// TwinCAT 3 PLC project PLC
// ProgramVersion: 3.1.4024.0
// libraries:
//   CmpBitmapPool, * (System)
//   Tc2_Standard, * (Beckhoff Automation GmbH)
//   Tc2_System, * (Beckhoff Automation GmbH)
//   Tc3_Module, * (Beckhoff Automation GmbH)
//   VisuDialogs, * (System)
//   VisuSymbols,3.5.10.0,System
// project tree:
//   DUTs/ CarPos.TcDUT
//   / GlobalTextList.TcGTLO, PlcTask.TcTTO
//   GVLs/ GVL.TcGVL
//   POUs/ CarHandle.TcPOU, MAIN.TcPOU
//   VISUs/ ImagePool.TcIPO (not stored), Visualization Manager.TcVMO (not stored), Visualization.TcVIS
// real-time tasks:
//   TASK PlcTask: cycle T#10ms, priority 20, ADS port 350

CONFIGURATION PLC
    RESOURCE PLC ON TwinCAT3
        TASK PlcTask(INTERVAL := T#10ms, PRIORITY := 20);
        PROGRAM MAIN WITH PlcTask : MAIN;
    END_RESOURCE
END_CONFIGURATION

// ---- DUTs/CarPos.TcDUT
TYPE CarPos :
STRUCT
// coordinates of car position in 3d parking
	X:	INT;
	Y:	INT;
	Z:	INT;
END_STRUCT
END_TYPE

// ---- GVLs/GVL.TcGVL
{attribute 'qualified_only'}
VAR_GLOBAL CONSTANT
	XPosMax		:	WORD:=2;
	YPosMax		:	WORD:=3;
	ZPosMax		:	WORD:=4;
END_VAR

// ---- POUs/MAIN.TcPOU
PROGRAM MAIN
VAR
	CarPlates		:	ARRAY [1..24] OF STRING(15) := ['AB12345', 'CD98765', 'EF24689', 'GH88888', 'IJ33388',
														'KL57483', 'MN35991', 'OP46819', 'RS00001', 'TU22229',
														'DE13578', 'ZX90909', 'YW10101', 'VW46372', 'ZZ00220',
														'WE00772', 'JK77001', 'PO39120', 'LW09126', 'RM01928',
														'EK11998', 'WY00664', 'HS05524', 'TT00099'];

	InsertCar		:	BOOL;					// insert car trigger
	
	FindCar			:	BOOL;					// find car trigger
	PlateToFind		:	STRING(15);				// car plate which should be found in the car park
	CarFoundPos		:	CarPos;					// position of found car
	
	RemoveCar		:	BOOL;					// remove car trigger
	CarToRemove		:	STRING(15);				// car plate which should be removed from the car park
	
	GetNoFreePlaces	:	BOOL;					// trigger for getting number of free places in car park
	
	rtAction		:	ARRAY[1..5] OF R_TRIG;
	FreePlaces		:	INT;
	
	CarHandle		:	CarHandle;
	
	Result			: 	BOOL;					// operation result
END_VAR

VAR RETAIN PERSISTENT
	CarPark			: ARRAY [1..GVL.XPosMax, 1..GVL.YPosMax, 1..GVL.ZPosMax] OF STRING(15);
	Idx				:	INT:=1;
END_VAR

CarHandle(ArrayPark:=CarPark);


rtAction[1](CLK:=InsertCar);
rtAction[2](CLK:=FindCar);
rtAction[3](CLK:=RemoveCar);
rtAction[4](CLK:=GetNoFreePlaces);

// insert car
IF rtAction[1].Q THEN
	Result := CarHandle.M_InsertCar(CarPlates[Idx]);
	FreePlaces := CarHandle.P_NumberFreePositions;
	Idx:= Idx + 1;
	IF Idx > 24 THEN 
		Idx := 1;
	END_IF
END_IF

// find car
IF rtAction[2].Q THEN
	Result := CarHandle.M_FindCar(CarPlate:=PlateToFind,FoundCarPos=>CarFoundPos);
END_IF

// delete car
IF rtAction[3].Q THEN
	Result := CarHandle.M_RemoveCar(CarPlate := CarToRemove);
	FreePlaces := CarHandle.P_NumberFreePositions;
END_IF

// get number of free places in car park
IF rtAction[4].Q THEN
	FreePlaces := CarHandle.P_NumberFreePositions;
END_IF

END_PROGRAM

// ---- POUs/CarHandle.TcPOU
FUNCTION_BLOCK CarHandle
VAR_INPUT
END_VAR
VAR_OUTPUT
END_VAR
VAR_IN_OUT
	ArrayPark		:	ARRAY[*,*,*] OF STRING(15);	// pointer to 3d array
END_VAR
VAR
	Loop			:	CarPos;						// temp. variable
	TotalPositions	: 	INT;						// total number of car positions in car park
END_VAR

(*
This FB handles three dimensional car park.
- ArrayPark - Dimension of the car park
*)


// copy ARRAY to local variables
Loop.X := DINT_TO_INT(UPPER_BOUND(ArrayPark,1));		// cordinate X
Loop.Y := DINT_TO_INT(UPPER_BOUND(ArrayPark,2));		// cordinate Y
Loop.Z := DINT_TO_INT(UPPER_BOUND(ArrayPark,3));		// cordinate Z

// total number of car positions in car park
TotalPositions := Loop.X * Loop.Y * Loop.Z;

METHOD M_FindCar : BOOL
VAR_INPUT
	CarPlate		:	STRING(15);		// plate number of the car
END_VAR
VAR
	CarPos			:	CarPos;			// location in car park
END_VAR
VAR_OUTPUT
	FoundCarPos		:	CarPos;			// location in car park
END_VAR
(*
This Method finds car in car park using its car plate.
CarPlate - car number plate which should be looked for in car park
Methods Returns TRUE if car was successfully found, otherwise FALSE
*)

// Loop over all position in the 3D car park
FOR CarPos.X:=1 TO Loop.X DO
	FOR CarPos.Y:=1 TO Loop.Y DO
		FOR CarPos.Z:=1 TO Loop.Z DO
			
			IF  FIND(ArrayPark[CarPos.X, CarPos.Y, CarPos.Z], CarPlate) > 0 THEN
				FoundCarPos := CarPos;	// copy coordinates where car was located
				M_FindCar := TRUE;
				RETURN;
			END_IF
			
		END_FOR
	END_FOR
END_FOR
M_FindCar := FALSE;
END_METHOD

METHOD M_InsertCar : BOOL
VAR_INPUT
	CarPlate		:	STRING(15);		// plate number of the car
END_VAR
VAR
	CarPos			:	CarPos;			// location in car park
END_VAR
(*
This Method inserts one car into car park.
CarPlate - car number plate which should be insert into car park
Methods Returns TRUE if car was successfully inserted, otherwise FALSE
*)

// Loop over all position in the 3D car park
FOR CarPos.X:=1 TO Loop.X DO
	FOR CarPos.Y:=1 TO Loop.Y DO
		FOR CarPos.Z:=1 TO Loop.Z DO
			
			// insert car at the first free location in the car park
			IF ArrayPark[CarPos.X, CarPos.Y, CarPos.Z]='' THEN
				ArrayPark[CarPos.X, CarPos.Y, CarPos.Z] := CarPlate;
				M_InsertCar := TRUE;
				RETURN;
			END_IF
			
		END_FOR
	END_FOR
END_FOR

M_InsertCar := FALSE;
END_METHOD

METHOD M_RemoveCar : BOOL
VAR_INPUT
	CarPlate		:	STRING(15);		// plate number of the car
END_VAR

VAR
	CarPos			:	CarPos;			// location in car park
END_VAR
(*
This Method removes one car in car park.
CarPlate - car number plate which should be removed in car park
Methods Returns TRUE if car was successfully removed, otherwise FALSE
*)

// Loop over all position in the 3D car park
FOR CarPos.X:=1 TO Loop.X DO
	FOR CarPos.Y:=1 TO Loop.Y DO
		FOR CarPos.Z:=1 TO Loop.Z DO
			
				IF FIND(ArrayPark[CarPos.X, CarPos.Y, CarPos.Z], CarPlate) > 0 THEN
					ArrayPark[CarPos.X, CarPos.Y, CarPos.Z]:=''; 	// remove car = set string empty 
					M_RemoveCar := TRUE;
					RETURN;
				END_IF
			
		END_FOR
	END_FOR
END_FOR

M_RemoveCar := TRUE;
END_METHOD

PROPERTY P_NumberFreePositions : INT

// Property returns number of free locations in car park
GET
VAR
	CarCount		: 	INT;			// number of occupied par places in car park
	CarPos			:	CarPos;			// location in car park
END_VAR
// Loop over all position in the 3D car park
FOR CarPos.X:=1 TO Loop.X DO
	FOR CarPos.Y:=1 TO Loop.Y DO
		FOR CarPos.Z:=1 TO Loop.Z DO
			
			IF ArrayPark[CarPos.X, CarPos.Y, CarPos.Z] <> '' THEN
				CarCount := CarCount+1;
			END_IF
			
		END_FOR
	END_FOR
END_FOR

P_NumberFreePositions := TotalPositions - CarCount;
END_GET
END_PROPERTY

END_FUNCTION_BLOCK

// ---- GlobalTextList.TcGTLO
TEXTLIST GlobalTextList
  316 = '%s'
  656 = '12387812'
  188 = 'Car Plate to Delete:'
  264 = 'Car PLate to Find:'
  432 = 'Car Plate to Find:'
  625 = 'Car to delete'
  296 = 'Car to Delete:'
  833 = 'Car to remove'
  597 = 'Car to Remove:'
  485 = 'Delete Car'
  174 = 'Find Car'
  267 = 'Found Car Position'
  242 = 'Insert Car'
  115 = 'Label'
  455 = 'Number of free places:\n\n%d'
  904 = 'Number of free places:\n%d'
  459 = 'Plate to delete'
  778 = 'Plate to find'
  298 = 'Plate to find: %s'
  396 = 'Remove Car'
  783 = 'Three Dimension Car Park'
  877 = 'X'
  615 = 'Y'
  950 = 'Z'
END_TEXTLIST

// ---- VISUs/Visualization.TcVIS
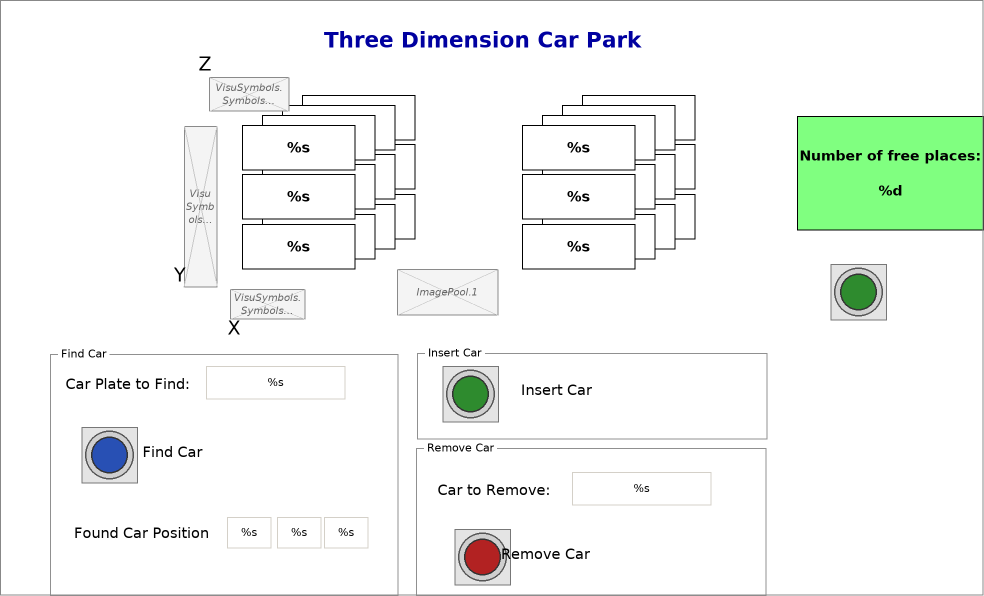
VISUALIZATION Visualization  // 984x596
    Rectangle (302,95 113x45), "%s", text variable: MAIN.CarPark[1,3,4], colour toggle: MAIN.CarPark[1,3,4] <> ''
    Rectangle (302,194 113x45), "%s", text variable: MAIN.CarPark[1,1,4], colour toggle: MAIN.CarPark[1,1,4] <> ''
    Rectangle (302,144 113x45), "%s", text variable: MAIN.CarPark[1,2,4], colour toggle: MAIN.CarPark[1,2,4] <> ''
    Rectangle (282,204 113x45), "%s", text variable: MAIN.CarPark[1,1,3], colour toggle: MAIN.CarPark[1,1,3] <> ''
    Rectangle (282,154 113x45), "%s", text variable: MAIN.CarPark[1,2,3], colour toggle: MAIN.CarPark[1,2,3] <> ''
    Rectangle (282,105 113x45), "%s", text variable: MAIN.CarPark[1,3,3], colour toggle: MAIN.CarPark[1,3,3] <> ''
    Rectangle (262,115 113x45), "%s", text variable: MAIN.CarPark[1,3,2], colour toggle: MAIN.CarPark[1,3,2] <> ''
    Rectangle (262,164 113x45), "%s", text variable: MAIN.CarPark[1,2,2], colour toggle: MAIN.CarPark[1,2,2] <> ''
    Rectangle (262,214 113x45), "%s", text variable: MAIN.CarPark[1,1,2], colour toggle: MAIN.CarPark[1,1,2] <> ''
    Rectangle (242,224 113x45), "%s", text variable: MAIN.CarPark[1,1,1], colour toggle: MAIN.CarPark[1,1,1] <> ''
    Rectangle (242,174 113x45), "%s", text variable: MAIN.CarPark[1,2,1], colour toggle: MAIN.CarPark[1,2,1] <> ''
    Rectangle (242,125 113x45), "%s", text variable: MAIN.CarPark[1,3,1], colour toggle: MAIN.CarPark[1,3,1] <> ''
    Rectangle (582,95 113x45), "%s", text variable: MAIN.CarPark[2,3,4], colour toggle: MAIN.CarPark[2,3,4] <> ''
    Rectangle (582,194 113x45), "%s", text variable: MAIN.CarPark[2,1,4], colour toggle: MAIN.CarPark[2,1,4] <> ''
    Rectangle (582,144 113x45), "%s", text variable: MAIN.CarPark[2,2,4], colour toggle: MAIN.CarPark[2,2,4] <> ''
    Rectangle (562,204 113x45), "%s", text variable: MAIN.CarPark[2,1,3], colour toggle: MAIN.CarPark[2,1,3] <> ''
    Rectangle (562,154 113x45), "%s", text variable: MAIN.CarPark[2,2,3], colour toggle: MAIN.CarPark[2,2,3] <> ''
    Rectangle (562,105 113x45), "%s", text variable: MAIN.CarPark[2,3,3], colour toggle: MAIN.CarPark[2,3,3] <> ''
    Rectangle (542,115 113x45), "%s", text variable: MAIN.CarPark[2,3,2], colour toggle: MAIN.CarPark[2,3,2] <> ''
    Rectangle (542,164 113x45), "%s", text variable: MAIN.CarPark[2,2,2], colour toggle: MAIN.CarPark[2,2,2] <> ''
    Rectangle (542,214 113x45), "%s", text variable: MAIN.CarPark[2,1,2], colour toggle: MAIN.CarPark[2,1,2] <> ''
    Rectangle (522,224 113x45), "%s", text variable: MAIN.CarPark[2,1,1], colour toggle: MAIN.CarPark[2,1,1] <> ''
    Rectangle (522,174 113x45), "%s", text variable: MAIN.CarPark[2,2,1], colour toggle: MAIN.CarPark[2,2,1] <> ''
    Rectangle (522,125 113x45), "%s", text variable: MAIN.CarPark[2,3,1], colour toggle: MAIN.CarPark[2,3,1] <> ''
    Label (319,22 328x36), "Three Dimension Car Park"
    GroupBox (50,346 348x250), "Find Car"
        Label (3,20 150x36), "Car Plate to Find:"
        Textfield (156,20 139x33), "%s", tooltip "Plate to find", text variable: MAIN.PlateToFind
            OnMouseClick: write the text variable via Edit
        PushSwitch (20,81 79x56), tooltip "Find Car", variable: MAIN.FindCar, behaviour: TAP, style: Switch-PushSwitch-Blue
        Label (72,88 101x36), "Find Car"
        Label (9,169 165x36), "Found Car Position"
        Textfield (177,171 44x31), "%s", tooltip "Plate to find", text variable: MAIN.CarFoundPos.X
            OnMouseClick: write the text variable via Edit
        Textfield (227,171 44x31), "%s", tooltip "Plate to find", text variable: MAIN.CarFoundPos.Y
            OnMouseClick: write the text variable via Edit
        Textfield (274,171 44x31), "%s", tooltip "Plate to find", text variable: MAIN.CarFoundPos.Z
            OnMouseClick: write the text variable via Edit
        PushSwitch (769,-82 79x56), tooltip "Find Car", variable: MAIN.FindCar, behaviour: TAP, style: Switch-PushSwitch-Green
    Rectangle (797,116 187x114), "Number of free places: %d", text variable: MAIN.FreePlaces
    GroupBox (416,440 350x156), "Remove Car"
        Label (3,32 150x36), "Car to Remove:"
        Textfield (156,32 139x33), "%s", tooltip "Car to remove", text variable: MAIN.CarToRemove
            OnMouseClick: write the text variable via Edit
        PushSwitch (27,89 79x56), tooltip "Remove Car", variable: MAIN.RemoveCar, behaviour: TAP, style: Switch-PushSwitch-Red
        Label (79,96 101x36), "Remove Car"
    GroupBox (417,345 350x94), "Insert Car"
        PushSwitch (14,21 79x56), tooltip "Insert Car", variable: MAIN.InsertCar, behaviour: TAP, style: Switch-PushSwitch-Green
        Label (89,27 101x36), "Insert Car"
    Image (397,269 101x46), image: ImagePool.1
    Image (230,289 75x30), image: VisuSymbols.Symbols.ArrowBoldRight
    Image (184,126 33x161), image: VisuSymbols.Symbols.ArrowBoldUp
    Image (209,77 80x34), image: VisuSymbols.Symbols.ArrowBoldRightUp
    Label (214,310 40x36), "X"
    Label (160,257 40x36), "Y"
    Label (185,46 40x36), "Z"
END_VISUALIZATION
